PROGRAM z_PRESS

(*-------------------------------------------------------------------------------------------------------*)
(*v070_Vent  Respiradero*)
Mc._03_PRESS.v070_Vent.xOpen:=_00_vent.z_xRespiradero;


(*-------------------------------------------------------------------------------------------------------*)
(*v071_Load  Carga presion*)
Mc._03_PRESS.v071_Load.xOpen:=_00_vent.z_xCargaPres;



(*-------------------------------------------------------------------------------------------------------*)
(*v074_Unload  Desgarga de presion*)
Mc._03_PRESS.v074_Unload.xOpen:=_00_vent.Z_xDescarga;

END_PROGRAM

(* stored: Version 1.1.0.1, ProductVersion 3.1.4024.10
   POU z_PRESS: Id {b27e6df5-f57f-411e-969d-e10cfe643960}, SpecialFunc None *)
